INTERFACE ITF_SensorDecoratorTest EXTENDS ITF_Sensor

METHOD SetContract
VAR_INPUT
	bIN: BOOL;
END_VAR
END_METHOD

END_INTERFACE

(* stored: Version 1.1.0.1
   Itf ITF_SensorDecoratorTest: Id {a0f2d16b-b657-44ae-a8cc-b4101f3dfa25}
   Method SetContract: Id {8f48095d-bf4c-4e86-8462-502e949f6b96} *)
